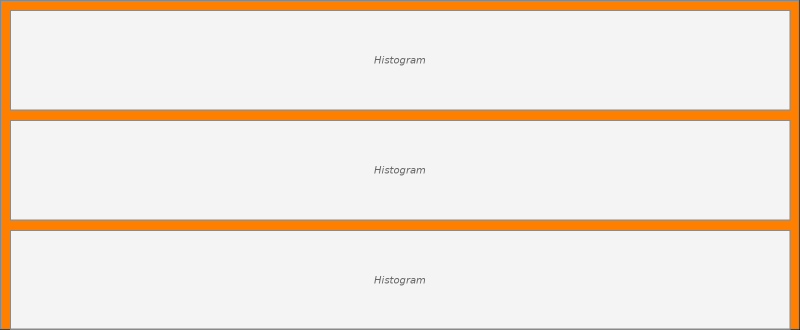
VISUALIZATION vPlotScreen  // 800x330
VAR_IN_OUT
	stControl : stControl;
	fbChamber	: fbChamber;
END_VAR
    Rectangle (0,0 800x330)
    Histogram (10,10 780x100), scale format: %.1f, scale 0..5
        p518627256: Bar
        p1518820177: fbChamber.arPlotPresure
        p102497268: fbChamber.arPlotPresure
        p788070771: ARRAY [0..1000] OF REAL
    Histogram (10,120 780x100), scale format: %.1f, scale 8..14
        p518627256: Volt
        p1518820177: fbChamber.arPlotVoltage
        p102497268: fbChamber.arPlotVoltage
        p788070771: ARRAY [0..1000] OF REAL
    Histogram (10,230 780x100), scale format: %.1f, scale 0..15
        p518627256: Amper
        p1518820177: fbChamber.arPlotCurrent
        p102497268: fbChamber.arPlotCurrent
        p788070771: ARRAY [0..1000] OF REAL
END_VISUALIZATION

(* stored: Version 1.1.0.1, ProductVersion 3.1.4024.12
   Visu vPlotScreen: Id {7e5ca3e9-13f3-4fa6-adb3-c62f6339811d} *)
